// TIA Portal V20 export
FUNCTION "sHREK" : Void   // FC1, LAD
{ S7_Optimized_Access := 'TRUE' }
// stored: SetENOAutomatically false
BEGIN
END_FUNCTION
